(* PLC project SafeLOGIC, BrAutomation SafeDESIGNER  5.24.1.0 *)
(* stored: companyURL http://www.br-automation.com, creationDateTime Sun Jun 29 13:11:13 2025 *)

PROGRAM Main
  VAR  (* added by the conversion: wires and edge detectors of the diagram *)
    _NOT_S80_OUT : ANY;
    _AND_S78_OUT : ANY;
  END_VAR

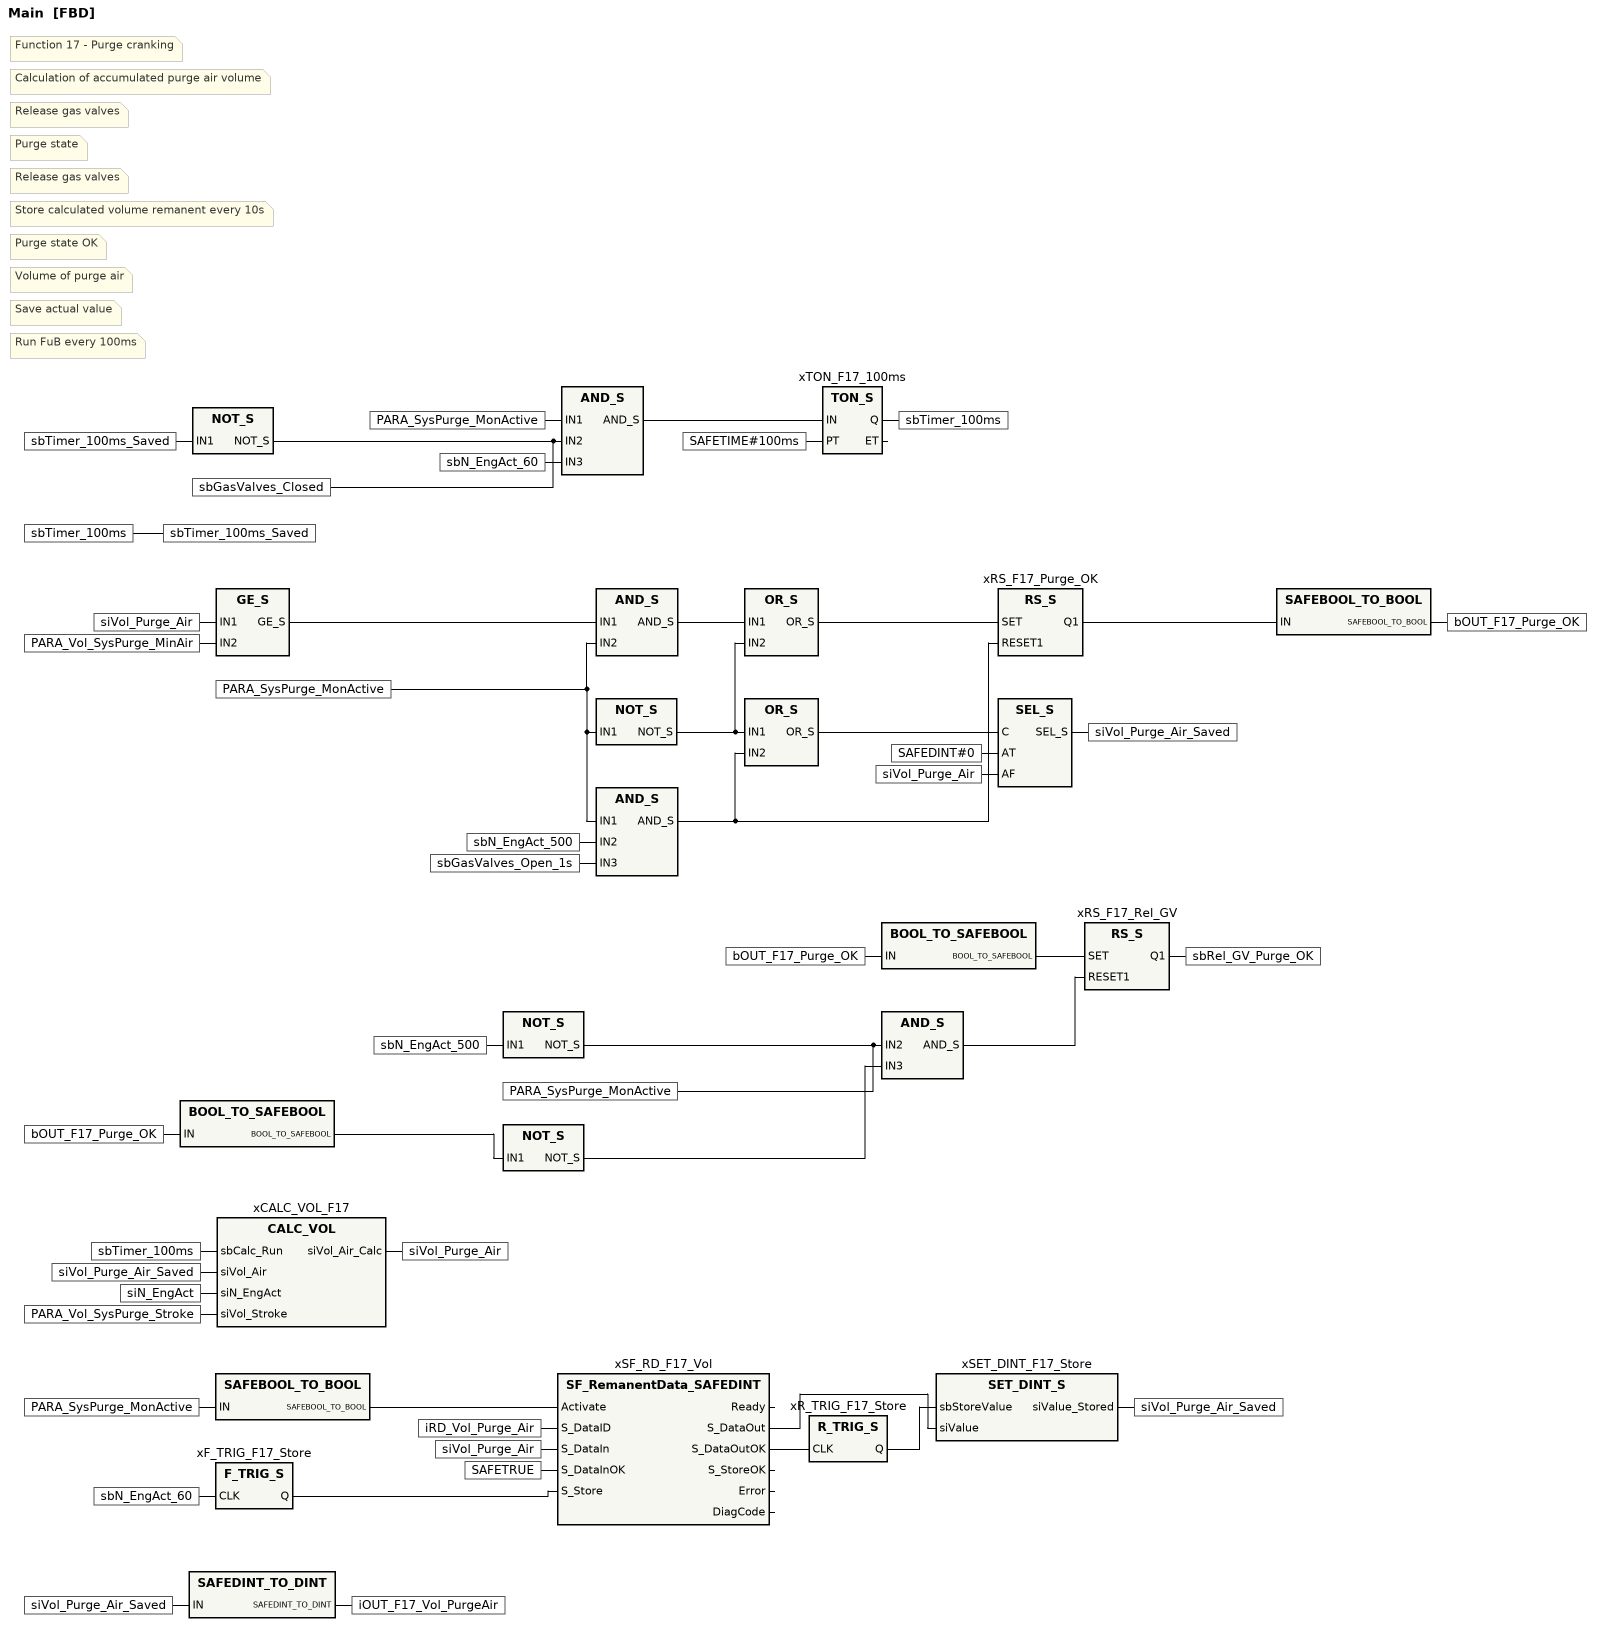
(* FBD diagram, written out as Structured Text *)
(* Function 17 - Purge cranking *)
(* Calculation of accumulated purge air volume *)
xTON_F17_100ms(IN := AND_S(PARA_SysPurge_MonActive, sbGasValves_Closed, sbN_EngAct_60, NOT_S(sbTimer_100ms_Saved)), PT := SAFETIME#100ms);
sbTimer_100ms := xTON_F17_100ms.Q;
(* Run FuB every 100ms *)
xCALC_VOL_F17(sbCalc_Run := sbTimer_100ms, siVol_Air := siVol_Purge_Air_Saved, siN_EngAct := siN_EngAct, siVol_Stroke := PARA_Vol_SysPurge_Stroke);
siVol_Purge_Air := xCALC_VOL_F17.siVol_Air_Calc;
(* Save actual value *)
sbTimer_100ms_Saved := sbTimer_100ms;
(* Purge state *)
(* Purge state OK *)
_NOT_S80_OUT := NOT_S(PARA_SysPurge_MonActive);
_AND_S78_OUT := AND_S(PARA_SysPurge_MonActive, sbN_EngAct_500, sbGasValves_Open_1s);
xRS_F17_Purge_OK(SET := OR_S(AND_S(GE_S(siVol_Purge_Air, PARA_Vol_SysPurge_MinAir), PARA_SysPurge_MonActive), _NOT_S80_OUT), RESET1 := _AND_S78_OUT);
bOUT_F17_Purge_OK := SAFEBOOL_TO_BOOL(xRS_F17_Purge_OK.Q1);
siVol_Purge_Air_Saved := SEL_S(OR_S(_NOT_S80_OUT, _AND_S78_OUT), SAFEDINT#0, siVol_Purge_Air);
(* Release gas valves *)
(* Release gas valves *)
xRS_F17_Rel_GV(SET := BOOL_TO_SAFEBOOL(bOUT_F17_Purge_OK), RESET1 := AND_S(PARA_SysPurge_MonActive, NOT_S(sbN_EngAct_500), NOT_S(BOOL_TO_SAFEBOOL(bOUT_F17_Purge_OK))));
sbRel_GV_Purge_OK := xRS_F17_Rel_GV.Q1;
(* Store calculated volume remanent every 10s *)
xF_TRIG_F17_Store(CLK := sbN_EngAct_60);
xSF_RD_F17_Vol(Activate := SAFEBOOL_TO_BOOL(PARA_SysPurge_MonActive), S_DataID := iRD_Vol_Purge_Air, S_DataIn := siVol_Purge_Air, S_DataInOK := SAFETRUE, S_Store := xF_TRIG_F17_Store.Q);
xR_TRIG_F17_Store(CLK := xSF_RD_F17_Vol.S_DataOutOK);
xSET_DINT_F17_Store(sbStoreValue := xR_TRIG_F17_Store.Q, siValue := xSF_RD_F17_Vol.S_DataOut);
siVol_Purge_Air_Saved := xSET_DINT_F17_Store.siValue_Stored;
(* Volume of purge air *)
iOUT_F17_Vol_PurgeAir := SAFEDINT_TO_DINT(siVol_Purge_Air_Saved);
END_PROGRAM
